// Mitsubishi GX Works2 project: exemplo ciclico   PLC: Q03UDV

PROGRAM MAIN
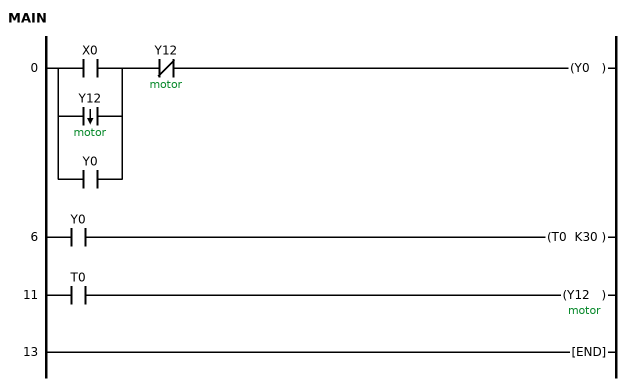
0     LD      X0
      ORF     Y12  ; motor
      OR      Y0
      ANI     Y12  ; motor
      OUT     Y0
6     LD      Y0
      OUT     T0 K30
11    LD      T0
      OUT     Y12  ; motor
13    END
END_PROGRAM
